// TIA Portal project "ParcelSortWithLinearAxises_1200" (V15.1)

(* hardware
DEVICE "S7-1200-Station_1"  S7-1200 Station
   slot 0: "Baugruppenträger_0"  S7-1200 Rack  Rack  V1.0
   slot 1: "PLC_1"  CPU 1214C AC/DC/Rly  6ES7 214-1BG40-0XB0  V4.2
   slot 2: "AI 4x13BIT/AQ 2x14BIT_1"  SM 1234 AI4/AQ2  6ES7 234-4HE30-0XB0  V1.0
*)

// ===== PLC "PLC_1"  CPU 1214C AC/DC/Rly =====

VAR_GLOBAL   // PLC tag table "Standard-Variablentabelle"
   "ControlOnFlag" AT %M0.0 : Bool;
   "Step1" AT %M0.1 : Bool;
   "Step2" AT %M0.2 : Bool;
   "Step3" AT %M0.3 : Bool;
   "Step4" AT %M0.4 : Bool;
   "Step5" AT %M0.5 : Bool;
   "Step6" AT %M0.6 : Bool;
   "StepActive" AT %M1.7 : Bool;
   "vertAxisEdgeFlag1" AT %M2.0 : Bool;
   "vertAxisEdgeFlag2" AT %M2.1 : Bool;
   "horizAxisEdgeFlag1" AT %M2.2 : Bool;
   "horizAxisEdgeFlag2" AT %M2.3 : Bool;
   "vertAxisEdgeFlag3" AT %M2.4 : Bool;
   "Step7" AT %M0.7 : Bool;
   "Step2A" AT %M1.0 : Bool;
   "Step9" AT %M1.1 : Bool;
   "vertAxisEdgeFlag4" AT %M2.5 : Bool;
   "horizAxisEdgeFlag3" AT %M2.6 : Bool;
   "horizAxisEdgeFlag4" AT %M2.7 : Bool;
   "vertAxisEdgeFlag5" AT %M3.0 : Bool;
   "GetYTargetPosIsOk" AT %M3.1 : Bool;
   "GetxTargetPosIsOk" AT %M3.2 : Bool;
   "B6ParcelGrapped" AT %E1.2 : Bool;
END_VAR

VAR_GLOBAL   // PLC tag table "Variablentabelle aus XML_1"
   "HorizontalAxisAbsPos" AT %IW2 : Word;
   "VerticalAxisAbsPos" AT %IW4 : Word;
   "P1ControlOn" AT %Q0.0 : Bool;
   "M1HorizAxis" AT %Q0.1 : Bool;
   "M2VertAxis" AT %Q0.2 : Bool;
   "HorizAxisGoToNewPos" AT %Q0.3 : Bool;
   "S1ControlOnPushButton" AT %I0.0 : Bool;
   "S2ControlOffPushButton" AT %I0.1 : Bool;   // NC
   "S3StartSort" AT %I0.2 : Bool;
   "B1ParcelInPos" AT %I0.3 : Bool;
   "B2HorizAxisMinPos" AT %I0.4 : Bool;   // NC
   "B3HorizAxisMaxPos" AT %I0.5 : Bool;   // NC
   "B4VertAxisMinPos" AT %I0.6 : Bool;   // NC
   "B5VertAxisMaxPos" AT %I0.7 : Bool;   // NC
   "HorizAxisNewPosReached" AT %I1.0 : Bool;
   "VertAxisNewPosReached" AT %I1.1 : Bool;
   "TargetStoragePlace" AT %IW6 : Word;
   "VertAxisGoToNewPos" AT %Q0.4 : Bool;
   "HorizAxisTargetPosAbs" AT %QW2 : Word;
   "VertAxisTargetPosAbs" AT %QW4 : Word;
   "VacuumOn" AT %Q0.5 : Bool;
END_VAR

// folder: System blocks/Program resources

DATA_BLOCK "ParcelGrappedTimer"   // DB1
{ S7_Optimized_Access := 'TRUE' }
AUTHOR : Simatic
FAMILY : IEC
NAME : IEC_TMR
VERSION : 1.0
// stored: InstanceOfName IEC_TIMER
"IEC_TIMER"
BEGIN
END_DATA_BLOCK

// folder: (top level)

FUNCTION "Steps" : Void   // FC1, FBD
{ S7_Optimized_Access := 'TRUE' }
VERSION : 0.1
   VAR_TEMP   // added for the SCL form of the ladder/FBD networks
      _w1 : Bool;
   END_VAR
BEGIN

REGION Network 1: wait for parcel
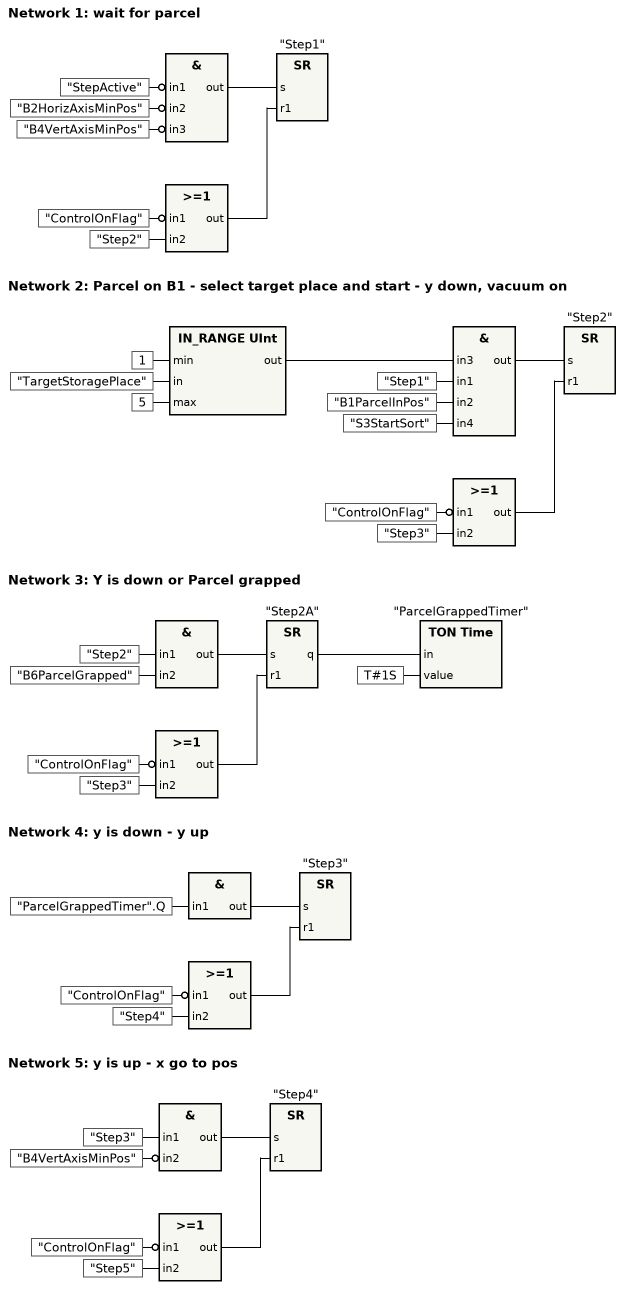
   IF NOT "StepActive" AND NOT "B2HorizAxisMinPos" AND NOT "B4VertAxisMinPos" THEN
       "Step1" := TRUE;   // SR flip-flop
   END_IF;
   IF NOT "ControlOnFlag" OR "Step2" THEN "Step1" := FALSE; END_IF;
END_REGION

REGION Network 2: Parcel on B1 - select target place and start - y down, vacuum on
   IF (1 <= "TargetStoragePlace") AND ("TargetStoragePlace" <= 5) AND "Step1" AND "B1ParcelInPos" AND "S3StartSort" THEN
       "Step2" := TRUE;   // SR flip-flop
   END_IF;
   IF NOT "ControlOnFlag" OR "Step3" THEN "Step2" := FALSE; END_IF;
END_REGION

REGION Network 3: Y is down or Parcel grapped
   IF "Step2" AND "B6ParcelGrapped" THEN
       "Step2A" := TRUE;   // SR flip-flop
   END_IF;
   IF NOT "ControlOnFlag" OR "Step3" THEN "Step2A" := FALSE; END_IF;
   "ParcelGrappedTimer".TON(IN := "Step2A", PT := T#1S);   // TON coil
END_REGION

REGION Network 4: y is down - y up
   IF "ParcelGrappedTimer".Q THEN
       "Step3" := TRUE;   // SR flip-flop
   END_IF;
   IF NOT "ControlOnFlag" OR "Step4" THEN "Step3" := FALSE; END_IF;
END_REGION

REGION Network 5: y is up - x go to pos
   IF "Step3" AND NOT "B4VertAxisMinPos" THEN
       "Step4" := TRUE;   // SR flip-flop
   END_IF;
   IF NOT "ControlOnFlag" OR "Step5" THEN "Step4" := FALSE; END_IF;
END_REGION

REGION Network 6: x pos reached - y down
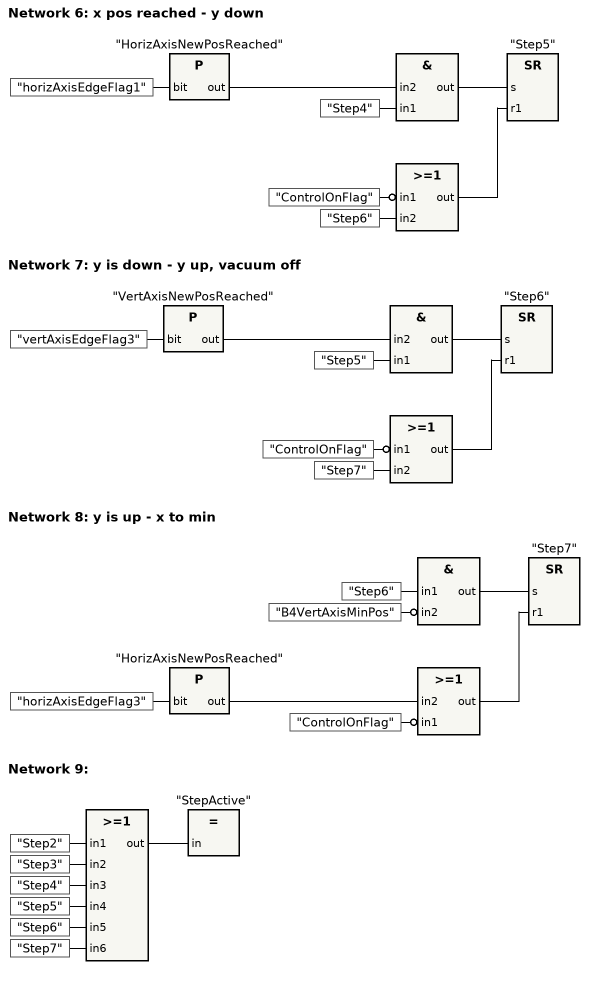
   #_w1 := "HorizAxisNewPosReached" AND NOT "horizAxisEdgeFlag1";   // rising edge of "HorizAxisNewPosReached"
   "horizAxisEdgeFlag1" := "HorizAxisNewPosReached";
   IF #_w1 AND "Step4" THEN
       "Step5" := TRUE;   // SR flip-flop
   END_IF;
   IF NOT "ControlOnFlag" OR "Step6" THEN "Step5" := FALSE; END_IF;
END_REGION

REGION Network 7: y is down - y up, vacuum off
   #_w1 := "VertAxisNewPosReached" AND NOT "vertAxisEdgeFlag3";   // rising edge of "VertAxisNewPosReached"
   "vertAxisEdgeFlag3" := "VertAxisNewPosReached";
   IF #_w1 AND "Step5" THEN
       "Step6" := TRUE;   // SR flip-flop
   END_IF;
   IF NOT "ControlOnFlag" OR "Step7" THEN "Step6" := FALSE; END_IF;
END_REGION

REGION Network 8: y is up - x to min
   #_w1 := "HorizAxisNewPosReached" AND NOT "horizAxisEdgeFlag3";   // rising edge of "HorizAxisNewPosReached"
   "horizAxisEdgeFlag3" := "HorizAxisNewPosReached";
   IF "Step6" AND NOT "B4VertAxisMinPos" THEN
       "Step7" := TRUE;   // SR flip-flop
   END_IF;
   IF #_w1 OR NOT "ControlOnFlag" THEN "Step7" := FALSE; END_IF;
END_REGION

REGION Network 9
   "StepActive" := "Step2" OR "Step3" OR "Step4" OR "Step5" OR "Step6" OR "Step7";
END_REGION
END_FUNCTION

FUNCTION "GetYTargetPos" : Void   // FC2, FBD
{ S7_Optimized_Access := 'TRUE' }
VERSION : 0.1
BEGIN

REGION Network 1
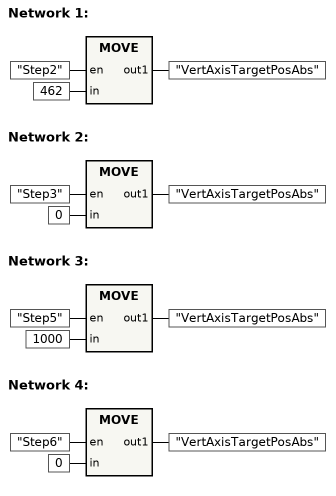
   IF "Step2" THEN "VertAxisTargetPosAbs" := 462; END_IF;
END_REGION

REGION Network 2
   IF "Step3" THEN "VertAxisTargetPosAbs" := 0; END_IF;
END_REGION

REGION Network 3
   IF "Step5" THEN "VertAxisTargetPosAbs" := 1000; END_IF;
END_REGION

REGION Network 4
   IF "Step6" THEN "VertAxisTargetPosAbs" := 0; END_IF;
END_REGION
END_FUNCTION

FUNCTION "Settings" : Void   // FC3, FBD
{ S7_Optimized_Access := 'TRUE' }
VERSION : 0.1
   VAR_TEMP   // added for the SCL form of the ladder/FBD networks
      _w1 : Bool;
   END_VAR
BEGIN

REGION Network 1
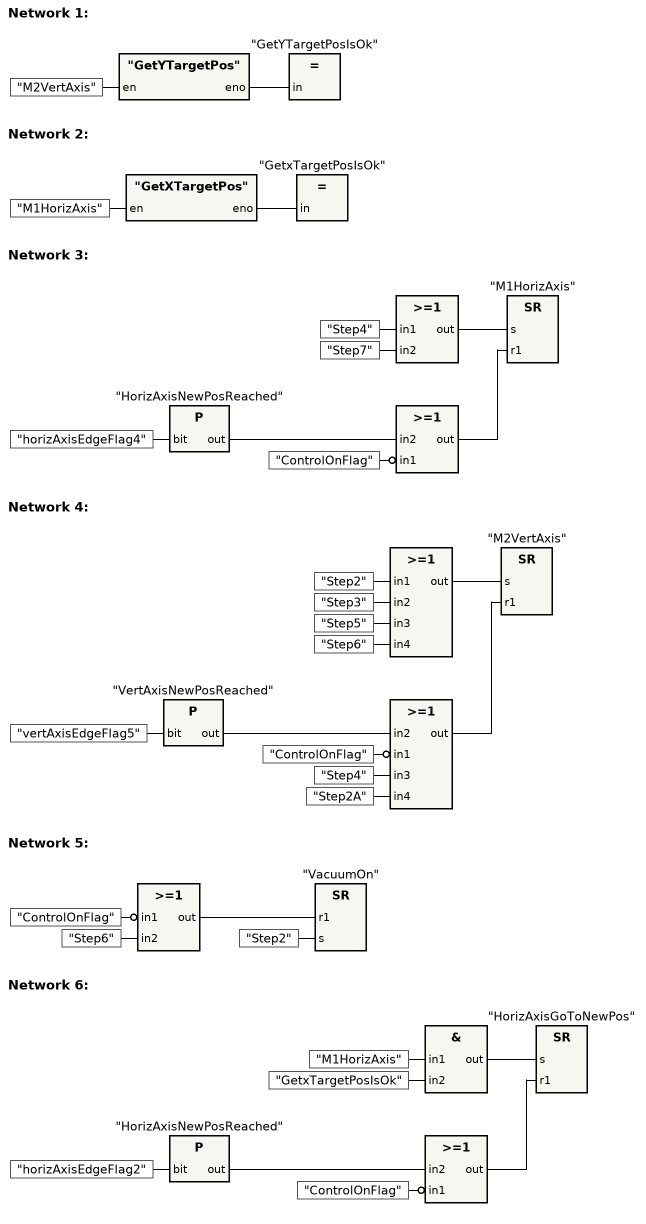
   "GetYTargetPos"(EN := "M2VertAxis", ENO => #_w1);
   "GetYTargetPosIsOk" := #_w1;
END_REGION

REGION Network 2
   "GetXTargetPos"(EN := "M1HorizAxis", ENO => #_w1);
   "GetxTargetPosIsOk" := #_w1;
END_REGION

REGION Network 3
   #_w1 := "HorizAxisNewPosReached" AND NOT "horizAxisEdgeFlag4";   // rising edge of "HorizAxisNewPosReached"
   "horizAxisEdgeFlag4" := "HorizAxisNewPosReached";
   IF "Step4" OR "Step7" THEN
       "M1HorizAxis" := TRUE;   // SR flip-flop
   END_IF;
   IF #_w1 OR NOT "ControlOnFlag" THEN "M1HorizAxis" := FALSE; END_IF;
END_REGION

REGION Network 4
   #_w1 := "VertAxisNewPosReached" AND NOT "vertAxisEdgeFlag5";   // rising edge of "VertAxisNewPosReached"
   "vertAxisEdgeFlag5" := "VertAxisNewPosReached";
   IF "Step2" OR "Step3" OR "Step5" OR "Step6" THEN
       "M2VertAxis" := TRUE;   // SR flip-flop
   END_IF;
   IF #_w1 OR NOT "ControlOnFlag" OR "Step4" OR "Step2A" THEN "M2VertAxis" := FALSE; END_IF;
END_REGION

REGION Network 5
   IF "Step2" THEN
       "VacuumOn" := TRUE;   // SR flip-flop
   END_IF;
   IF NOT "ControlOnFlag" OR "Step6" THEN "VacuumOn" := FALSE; END_IF;
END_REGION

REGION Network 6
   #_w1 := "HorizAxisNewPosReached" AND NOT "horizAxisEdgeFlag2";   // rising edge of "HorizAxisNewPosReached"
   "horizAxisEdgeFlag2" := "HorizAxisNewPosReached";
   IF "M1HorizAxis" AND "GetxTargetPosIsOk" THEN
       "HorizAxisGoToNewPos" := TRUE;   // SR flip-flop
   END_IF;
   IF #_w1 OR NOT "ControlOnFlag" THEN "HorizAxisGoToNewPos" := FALSE; END_IF;
END_REGION

REGION Network 7
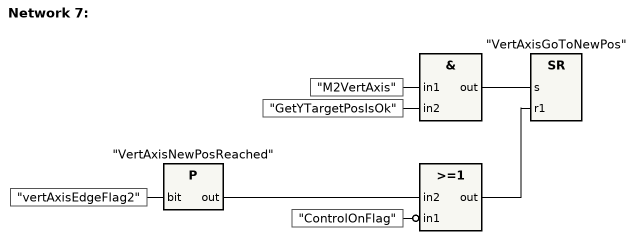
   #_w1 := "VertAxisNewPosReached" AND NOT "vertAxisEdgeFlag2";   // rising edge of "VertAxisNewPosReached"
   "vertAxisEdgeFlag2" := "VertAxisNewPosReached";
   IF "M2VertAxis" AND "GetYTargetPosIsOk" THEN
       "VertAxisGoToNewPos" := TRUE;   // SR flip-flop
   END_IF;
   IF #_w1 OR NOT "ControlOnFlag" THEN "VertAxisGoToNewPos" := FALSE; END_IF;
END_REGION
END_FUNCTION

FUNCTION "GetXTargetPos" : Void   // FC4, FBD
{ S7_Optimized_Access := 'TRUE' }
VERSION : 0.1
   VAR_TEMP
      TempTargetPosNumber : UInt;
   END_VAR
BEGIN

REGION Network 1
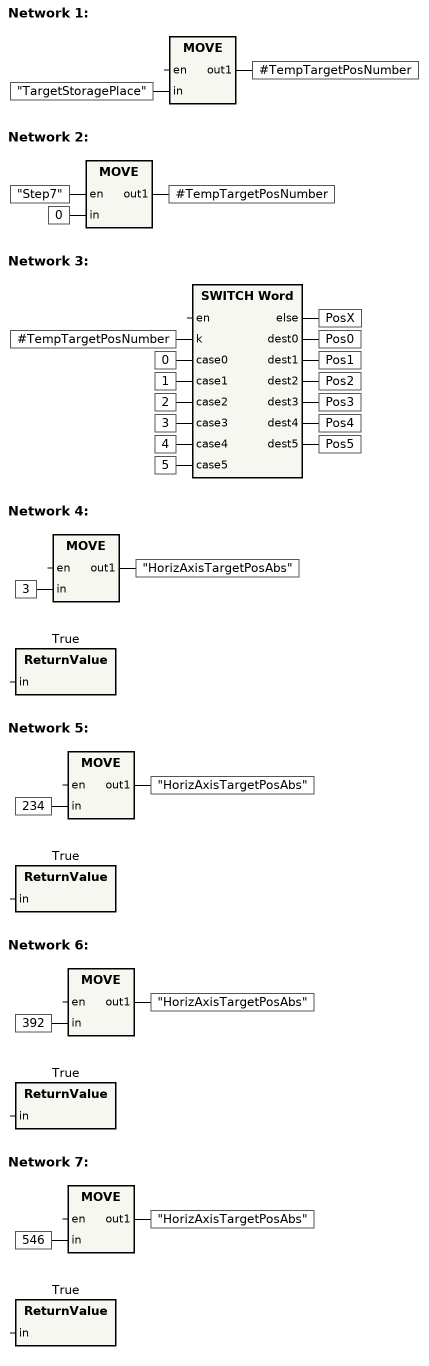
   #TempTargetPosNumber := "TargetStoragePlace";
END_REGION

REGION Network 2
   IF "Step7" THEN #TempTargetPosNumber := 0; END_IF;
END_REGION

REGION Network 3
   // no SCL statement known for Switch: written as a call
   Switch(k := #TempTargetPosNumber,
          case0 := 0,
          case1 := 1,
          case2 := 2,
          case3 := 3,
          case4 := 4,
          case5 := 5,
          "else" => PosX,
          dest0 => Pos0,
          dest1 => Pos1,
          dest2 => Pos2,
          dest3 => Pos3,
          dest4 => Pos4,
          dest5 => Pos5);
END_REGION

REGION Network 4
   Pos0:
   "HorizAxisTargetPosAbs" := 3;
   ENO := True;
   RETURN;
END_REGION

REGION Network 5
   Pos1:
   "HorizAxisTargetPosAbs" := 234;
   ENO := True;
   RETURN;
END_REGION

REGION Network 6
   Pos2:
   "HorizAxisTargetPosAbs" := 392;
   ENO := True;
   RETURN;
END_REGION

REGION Network 7
   Pos3:
   "HorizAxisTargetPosAbs" := 546;
   ENO := True;
   RETURN;
END_REGION

REGION Network 8
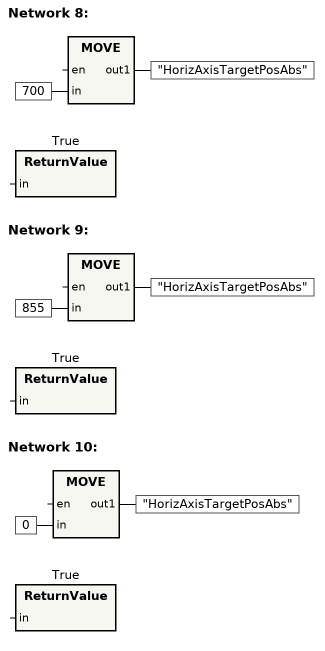
   Pos4:
   "HorizAxisTargetPosAbs" := 700;
   ENO := True;
   RETURN;
END_REGION

REGION Network 9
   Pos5:
   "HorizAxisTargetPosAbs" := 855;
   ENO := True;
   RETURN;
END_REGION

REGION Network 10
   PosX:
   "HorizAxisTargetPosAbs" := 0;
   ENO := True;
   RETURN;
END_REGION
END_FUNCTION

FUNCTION "MHJ-PLC-Lab-Function-S71200" : Void   // FC9000, SCL
{ S7_Optimized_Access := 'TRUE' }
VERSION : 0.1
   VAR_TEMP
      rdTimeReturn : Int;
      outputTime : DTL;
      SyncVal : Byte;
      forVal : Int;
      forVal_2 : Int;
      Value : Byte;
   END_VAR
   VAR CONSTANT
      CompVal : Byte := 16#34;
      Value_01 : Byte := 16#11;
      Value_01_DW : DWord := 16#A165_D992;
      Value_02_DW : DWord := 16#58BE_4401;
   END_VAR
BEGIN

   #Value:=PEEK(area := 16#82,
        dbNumber := 0,
        byteOffset := 511);
   #Value := #Value + 1;

   POKE(area := 16#82,
        dbNumber := 0,
        byteOffset := 511,
        value := #Value);

   POKE(area:=16#81,
        dbNumber:=0,
        byteOffset:=1016,
        value:=#Value_01_DW);
   POKE(area := 16#81,
        dbNumber := 0,
        byteOffset := 1020,
        value := #Value_02_DW);

   POKE(area := 16#81,
        dbNumber := 0,
        byteOffset := 511,
        value := B#16#00);

   FOR #forVal := 0 TO 120 DO
       FOR #forVal_2:=0 TO 10 DO
           #rdTimeReturn:=RD_SYS_T(#outputTime);
           #rdTimeReturn := WR_SYS_T(#outputTime);
           #rdTimeReturn := RD_SYS_T(#outputTime);
           #rdTimeReturn := WR_SYS_T(#outputTime);
       END_FOR;
       #SyncVal:= PEEK(area := 16#81,
                      dbNumber := 0,
                      byteOffset := 511);
       IF #SyncVal = #CompVal THEN
          GOTO M_1;
       END_IF;
   END_FOR;
   RETURN;

   M_1:
   POKE(area := 16#81,
        dbNumber := 0,
        byteOffset := 511,
        value := B#16#0);
END_FUNCTION

ORGANIZATION_BLOCK "Main"   // OB1, FBD, ProgramCycle
TITLE = "Main Program Sweep (Cycle)"
{ S7_Optimized_Access := 'TRUE' }
VERSION : 0.1
   VAR_INPUT
      Initial_Call : Bool;   // Initial call of this OB
      Remanence : Bool;   // =True, if remanent data are available
   END_VAR
BEGIN

REGION Network 1
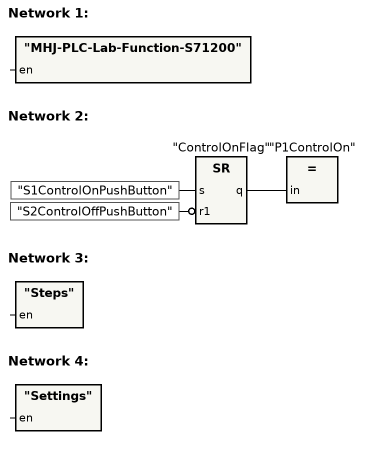
   "MHJ-PLC-Lab-Function-S71200"();
END_REGION

REGION Network 2
   IF "S1ControlOnPushButton" THEN
       "ControlOnFlag" := TRUE;   // SR flip-flop
   END_IF;
   IF NOT "S2ControlOffPushButton" THEN "ControlOnFlag" := FALSE; END_IF;
   "P1ControlOn" := "ControlOnFlag";
END_REGION

REGION Network 3
   "Steps"();
END_REGION

REGION Network 4
   "Settings"();
END_REGION
END_ORGANIZATION_BLOCK